Omron CX-Programmer project NewProject (CX-Programmer 9.81)

# PLC NewPLC1: CJ1M CPU11

## Global symbols (name address type ; comment)
0 CHANNEL  ; flag

## Program NewProgram1 (cyclic task 0)
Local symbols
b_start 0.00 BOOL
etapa_0 2.00 BOOL
etapa_1 2.01 BOOL  ; etapa 1 grafcet
etapa_2 2.02 BOOL  ; etapa 2 grafcet
flag_t1 T0001 BOOL  ; flag do temporizador 1
km1 100.00 BOOL  ; ligar km1
t_1 1 NUMBER  ; temporizador 1
tempo_t1 #50 NUMBER  ; tempo do temporizador 1

### Section Main

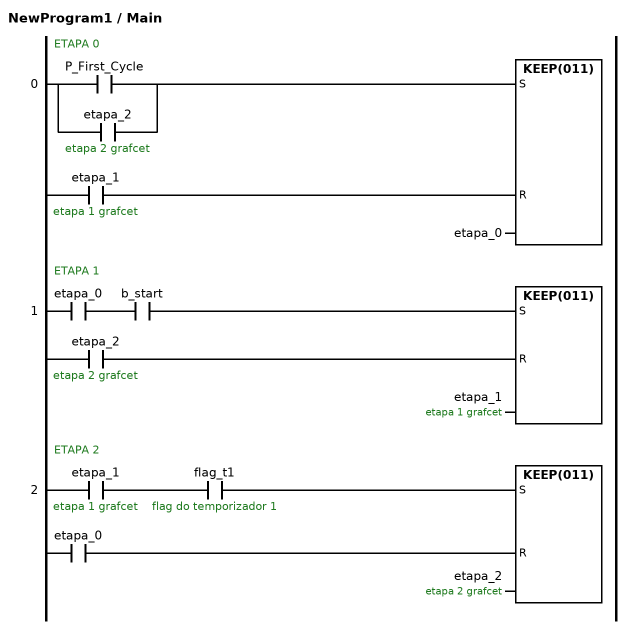
; rung 0: ETAPA 0
LD P_First_Cycle
OR etapa_2  ; etapa 2 grafcet
LD etapa_1  ; etapa 1 grafcet
KEEP(011) etapa_0
; rung 1: ETAPA 1
LD etapa_0
AND b_start
LD etapa_2  ; etapa 2 grafcet
KEEP(011) etapa_1  ; etapa 1 grafcet
; rung 2: ETAPA 2
LD etapa_1  ; etapa 1 grafcet
AND flag_t1  ; flag do temporizador 1
LD etapa_0
KEEP(011) etapa_2  ; etapa 2 grafcet

### Section Timers

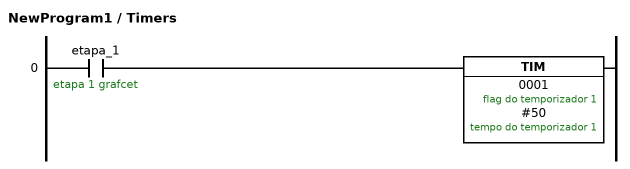
; rung 0
LD etapa_1  ; etapa 1 grafcet
TIM 0001 #50  ; tempo do temporizador 1, flag do temporizador 1

### Section OUT

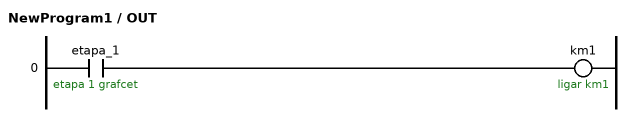
; rung 0
LD etapa_1  ; etapa 1 grafcet
OUT km1  ; ligar km1

### Section END
; rung 0
END(001)